FUNCTION_BLOCK FB_Pump_Simulator EXTENDS FB_Pump
VAR_INPUT
END_VAR
VAR_OUTPUT
    hydrualicPump_output : ST_Pump_Output;
END_VAR
VAR
END_VAR



ExecuteState();
IF NOT (nextState = curState)THEN
    StateTransition();
END_IF

ACTION ExecuteState:


CASE curState OF
	eState_Idle: ExecuteState_Idle();
	eState_Startup: ExecuteState_Startup();
	eState_Running: ExecuteState_Running();
	eState_Complete: ExecuteState_Complete();
    eState_Stopping: ExecuteState_Stopping();
    eState_Stopped: ExecuteState_Stopped();
	eState_Error: ExecuteState_Error();
	eState_Independent: ExecuteState_Independent();
END_CASE
END_ACTION

ACTION ExecuteState_Complete:

END_ACTION

ACTION ExecuteState_Error:
// Set Outputs
hydrualicPump_output.On := FALSE;
END_ACTION

ACTION ExecuteState_Idle:
// Set Outputs
hydrualicPump_output.On := FALSE;
END_ACTION

ACTION ExecuteState_Independent:
// Set Outputs
hydrualicPump_output.On := FALSE;
END_ACTION

ACTION ExecuteState_Running:
// Set Outputs
hydrualicPump_output.On := TRUE;
END_ACTION

ACTION ExecuteState_Startup:

// reset timers

// set output to true
nextState := eState_Running;
END_ACTION

ACTION ExecuteState_Stopped:
nextState := eState_Idle;
END_ACTION

ACTION ExecuteState_Stopping:
nextState := eState_Stopped;
END_ACTION

METHOD reset : BOOL
resetAlarms();

IF curState = eState_Complete THEN
	nextState := eState_Idle;
	reset := TRUE;
ELSIF curState = eState_Error THEN
    nextState := eState_Idle;
ELSE
	reset := FALSE;
END_IF
END_METHOD

METHOD start: BOOL
VAR_INPUT
END_VAR
IF curState = eState_Idle THEN
	nextState := eState_Startup;
	start := TRUE;
ELSE
	start := FALSE;
END_IF
END_METHOD

ACTION StateTransition:
SUPER^.StateTransition();
END_ACTION

END_FUNCTION_BLOCK

(* stored: Version 1.1.0.1, ProductVersion 3.1.4024.9
   POU FB_Pump_Simulator: Id {81a1403c-06b9-44cf-be98-10fc56b4a99a}, SpecialFunc None
   Folder StateMachine: Id {6591b63e-7203-44ce-98c9-3c70bf047d96}
   Folder States: Id {412a3bdd-03bd-4fac-8969-2dc0f12d5280}
   Action ExecuteState: Id {90abc579-3786-4c63-8fb8-91241bbea807}
   Action ExecuteState_Complete: Id {f93f4aec-57d3-475c-9289-7867fedfa70e}
   Action ExecuteState_Error: Id {b4eb4842-456b-45f9-a1c3-b94c107a69d7}
   Action ExecuteState_Idle: Id {0399335e-4015-4def-9a68-60423b4478fc}
   Action ExecuteState_Independent: Id {4bf016da-0110-4136-8caa-2802db38d79f}
   Action ExecuteState_Running: Id {ac20075c-10e2-4943-bab1-0f12573d34ba}
   Action ExecuteState_Startup: Id {abcfa1d4-34b0-46b6-8c91-a9afbaa12c93}
   Action ExecuteState_Stopped: Id {67797a12-7c77-4492-ab10-ec3190001a05}
   Action ExecuteState_Stopping: Id {325aea95-89d3-4005-8979-9ede55652c3e}
   Method reset: Id {1b213662-a46b-47c9-aca3-379bff81390e}
   Method start: Id {15844ad4-1357-413d-a2ba-05ff496a7bbd}
   Action StateTransition: Id {43b8d4fe-c0dc-4a47-ae35-439203a69ee1} *)
